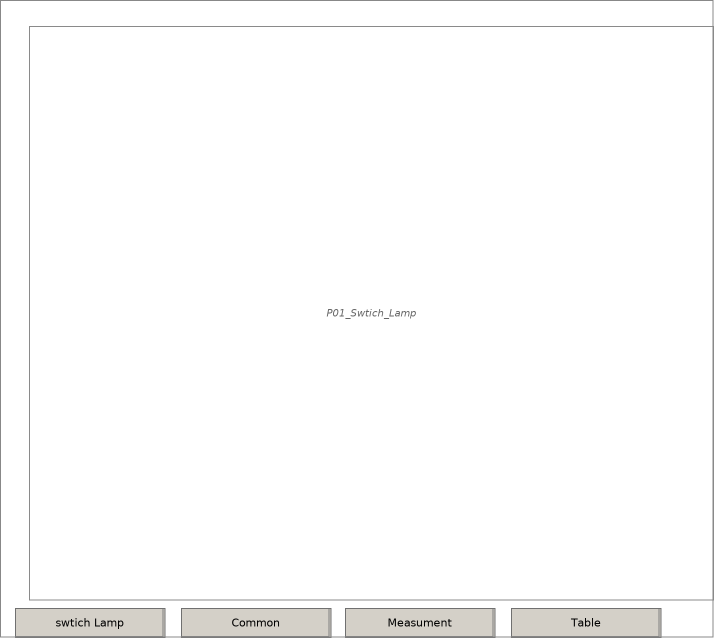
VISUALIZATION P00_Main  // 714x638
    Button (15,608 150x30), "swtich Lamp"
        OnMouseDown: FrameSelectionChange Selection=SelectedFrame=647e187a-0755-4409-bbed-ce6851db0410, GlobSel=AssignType=Directly, SelType=Locally
    Frame (29,26 685x574)
        shows P01_Swtich_Lamp()
        shows P02_Measurement()
        shows P03_Common()
        shows P04_Table()
    Button (181,608 150x30), "Common"
        OnMouseDown: FrameSelectionChange Selection=SelectedFrame=647e187a-0755-4409-bbed-ce6851db0410, Selection=2, GlobSel=AssignType=Directly, SelType=Locally
    Button (345,608 150x30), "Measument"
        OnMouseDown: FrameSelectionChange Selection=SelectedFrame=647e187a-0755-4409-bbed-ce6851db0410, Selection=1, GlobSel=AssignType=Directly, SelType=Locally
    Button (511,608 150x30), "Table"
        OnMouseDown: FrameSelectionChange Selection=SelectedFrame=647e187a-0755-4409-bbed-ce6851db0410, Selection=3, GlobSel=AssignType=Directly, SelType=Locally
END_VISUALIZATION

(* stored: Version 1.1.0.1, ProductVersion 3.1.4024.6
   Visu P00_Main: Id {f173ba27-0cfe-48c4-a09e-5320b4276209} *)
